// Mitsubishi GX Works2 project: PLS_PLF   PLC: Q03UDV

PROGRAM MAIN
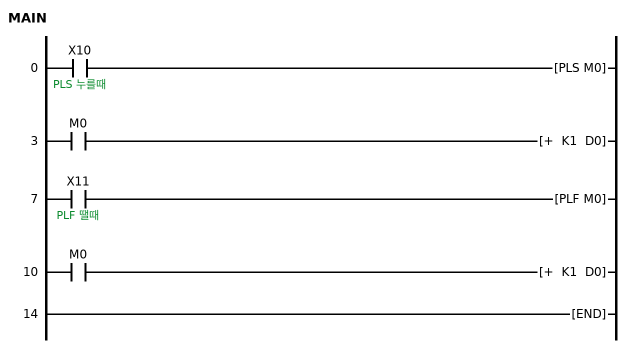
0     LD      X10  ; PLS 누를때
      PLS     M0
3     LD      M0
      +       K1 D0
7     LD      X11  ; PLF 땔때
      PLF     M0
10    LD      M0
      +       K1 D0
14    END
END_PROGRAM
